Staubli VAL3: processList.dtx

num nIndex
num nKey
num nRefresh
num nTime = 1
num nView
string sEvent
public string sItems
string sList
string sMenu[8]
string sMessage
string sType[3]
  [0] = "START Process"
  [1] = "MAIN Process"
  [2] = "END Process"
string sMenu8[8]
string sWrite
bool bButton[8]
bool bLarge
